INTERFACE ITF_BaseHMITopElement_View EXTENDS ITF_BaseHMIComponent_View

END_INTERFACE

(* stored: Version 1.1.0.1
   Itf ITF_BaseHMITopElement_View: Id {02116d65-3c4f-0345-19e7-8c8d9b7515ea} *)
